(* CODESYS project FunctionBlockExport.export

Project tree, tasks and I/O mapping:
  program Main [ST]
  function block Motor [ST]
*)

// Main
PROGRAM Main
VAR
	MyMotorInstance1 : Motor;
	MyMotorInstance2 : Motor;
	MyMotorInstance3 : Motor;
END_VAR


MyMotorInstance1();
MyMotorInstance2();
MyMotorInstance3();

END_PROGRAM

// Motor
FUNCTION_BLOCK PUBLIC Motor
VAR_INPUT
END_VAR
VAR_OUTPUT
END_VAR
VAR
END_VAR


// Motor control logic here

END_FUNCTION_BLOCK
